FUNCTION_BLOCK BYPASS_AX (* Bypass FB *)
  (* Standard: 61499-2 *)
  (* Version 1.0, 2026-05-07, franz *)
  PACKAGE logiBUS::signalprocessing::bypass;
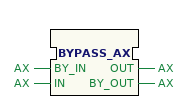
  SOCKETS
    BY_IN : adapter::types::unidirectional::AX; (* Bypass in *)
    IN : adapter::types::unidirectional::AX; (* Signal Input *)
  END_SOCKETS
  PLUGS
    OUT : adapter::types::unidirectional::AX; (* Signal Output *)
    BY_OUT : adapter::types::unidirectional::AX; (* Bypass out *)
  END_PLUGS
END_FUNCTION_BLOCK
